// TIA Portal V16 export
// export: Created 2024-05-13T12:48:19.9116386Z, ExportSetting WithDefaults, DisplayName Totally Integrated Automation Portal, DisplayVersion V16 Update 6, DisplayName TIA Portal Version Control Interface, DisplayVersion V16 Update 2, DisplayName TIA Portal Openness, DisplayVersion V16 Update 6, DisplayName TIA Portal Test Suite Advanced, DisplayVersion V16, DisplayName SINAMICS Startdrive Advanced, DisplayVersion V16 Update 5, DisplayName SINAMICS Startdrive G130, G150, S120, S150, SINAMICS MV, S210, DisplayVersion V16 Update 5, DisplayName SINAMICS Startdrive G110M, G120, G120C, G120D, G120P, G115D, DisplayVersion V16 Update 5, DisplayName STEP 7 Professional, DisplayVersion V16 Update 6, DisplayName STEP 7 Safety, DisplayVersion V16, DisplayName WinCC Advanced, DisplayVersion V16 Update 6
TYPE "SCA_inkjetMarker_flags"
// stored: IsFailsafeCompliant false
   STRUCT
      Speed_1 : Bool;   // Speed selection 1
      Speed_2 : Bool;   // Speed selection 2
      Speed_3 : Bool;   // Speed selection 3
      Speed_4 : Bool;   // Speed selection 4
      Trigger_on_p : Bool;   // Barcode reader trigger on
      Trigger_off_p : Bool;   // Barcode reader trigger off
      Device_stopped : Bool;
      Send_data : Bool;   // Send data to printer
      Print_data : Bool;   // Print data from printer
      Reading_done : Bool;   // Roll barcode reading done
      "Head fwd" : Bool;
      "Head left" : Bool;
   END_STRUCT;
END_TYPE
